// TIA Portal project "P6" (V17)

(* hardware
DEVICE "S7-1500/ET200MP station_1"  S7-1500 station
   slot 0: "Rail_0"  Rack  6ES7 590-1***0-0AA0
   slot 1: "PLC_1"  CPU 1515-2 PN  6ES7 515-2AM02-0AB0  V2.9
      slot 3: "CPU display_1"  6ES7591-1BA00-0AA0
      slot 32768: "PROFINET interface_1"  X1
         slot 32769: "Port_1"  X1 P1
         slot 32770: "Port_2"  X1 P2
      slot 33024: "PROFINET interface_2"  X2
         slot 33025: "Port_1"  X2 P1
      slot 34817: "Virtual CP interface port_1"  Virtual CP interface port  Virtual CP interface port
*)

// ===== PLC "PLC_1"  CPU 1515-2 PN =====

VAR_GLOBAL   // PLC tag table "Default tag table"
   "FWD PB" AT %I0.0 : Bool;
   "REV PB" AT %I0.1 : Bool;
   "MOTOR STOP" AT %I0.2 : Bool;
   "MOTOR TRIP" AT %I0.3 : Bool;
   "MOTOR FORWARD COIL" AT %Q0.0 : Bool;
   "MOTOR REVERSE COIL" AT %Q0.1 : Bool;
END_VAR

ORGANIZATION_BLOCK "Main"   // OB1, LAD, ProgramCycle
TITLE = "Main Program Sweep (Cycle)"
{ S7_Optimized_Access := 'TRUE' }
VERSION : 0.1
   VAR_INPUT
      Initial_Call : Bool;   // Initial call of this OB
      Remanence : Bool;   // =True, if remanent data are available
   END_VAR
BEGIN

REGION Network 1
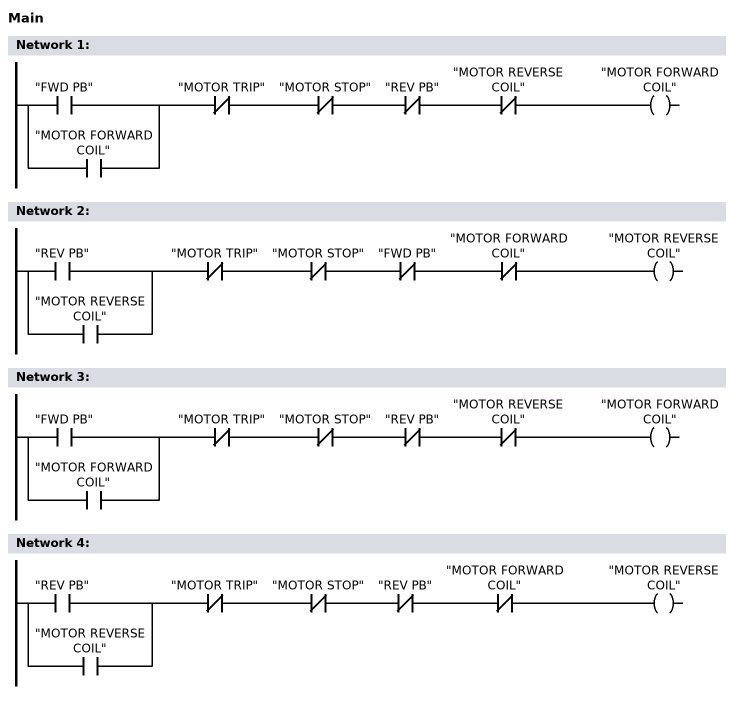
   RUNG wire#powerrail
      Contact( "FWD PB" )
      wire#w1
      I_Contact( "MOTOR TRIP" )
      I_Contact( "MOTOR STOP" )
      I_Contact( "REV PB" )
      I_Contact( "MOTOR REVERSE COIL" )
      Coil( "MOTOR FORWARD COIL" )
   END_RUNG
   RUNG wire#powerrail
      Contact( "MOTOR FORWARD COIL" )
   END_RUNG wire#w1
   // the same network as SCL:
   "MOTOR FORWARD COIL" := ("FWD PB" OR "MOTOR FORWARD COIL") AND NOT "MOTOR TRIP" AND NOT "MOTOR STOP" AND NOT "REV PB" AND NOT "MOTOR REVERSE COIL";
END_REGION

REGION Network 2
   RUNG wire#powerrail
      Contact( "REV PB" )
      wire#w1
      I_Contact( "MOTOR TRIP" )
      I_Contact( "MOTOR STOP" )
      I_Contact( "FWD PB" )
      I_Contact( "MOTOR FORWARD COIL" )
      Coil( "MOTOR REVERSE COIL" )
   END_RUNG
   RUNG wire#powerrail
      Contact( "MOTOR REVERSE COIL" )
   END_RUNG wire#w1
   // the same network as SCL:
   "MOTOR REVERSE COIL" := ("REV PB" OR "MOTOR REVERSE COIL") AND NOT "MOTOR TRIP" AND NOT "MOTOR STOP" AND NOT "FWD PB" AND NOT "MOTOR FORWARD COIL";
END_REGION

REGION Network 3
   RUNG wire#powerrail
      Contact( "FWD PB" )
      wire#w1
      I_Contact( "MOTOR TRIP" )
      I_Contact( "MOTOR STOP" )
      I_Contact( "REV PB" )
      I_Contact( "MOTOR REVERSE COIL" )
      Coil( "MOTOR FORWARD COIL" )
   END_RUNG
   RUNG wire#powerrail
      Contact( "MOTOR FORWARD COIL" )
   END_RUNG wire#w1
   // the same network as SCL:
   "MOTOR FORWARD COIL" := ("FWD PB" OR "MOTOR FORWARD COIL") AND NOT "MOTOR TRIP" AND NOT "MOTOR STOP" AND NOT "REV PB" AND NOT "MOTOR REVERSE COIL";
END_REGION

REGION Network 4
   RUNG wire#powerrail
      Contact( "REV PB" )
      wire#w1
      I_Contact( "MOTOR TRIP" )
      I_Contact( "MOTOR STOP" )
      I_Contact( "REV PB" )
      I_Contact( "MOTOR FORWARD COIL" )
      Coil( "MOTOR REVERSE COIL" )
   END_RUNG
   RUNG wire#powerrail
      Contact( "MOTOR REVERSE COIL" )
   END_RUNG wire#w1
   // the same network as SCL:
   "MOTOR REVERSE COIL" := ("REV PB" OR "MOTOR REVERSE COIL") AND NOT "MOTOR TRIP" AND NOT "MOTOR STOP" AND NOT "REV PB" AND NOT "MOTOR FORWARD COIL";
END_REGION
END_ORGANIZATION_BLOCK